// TIA Portal project "Project1" (V17)

(* hardware
DEVICE "S7-1200 station_1"  S7-1200 Station
   slot 0: "Rack_0"  S7-1200 Rack  Rack  V1.0
   slot 1: "PLC_1"  CPU 1214C DC/DC/DC  6ES7 214-1AG31-0XB0  V3.0
   slot 3: "AQ 1x12BIT_1"  AQ1 signal board  6ES7 232-4HA30-0XB0  V1.0
*)

// ===== PLC "PLC_1"  CPU 1214C DC/DC/DC =====

VAR_GLOBAL   // PLC tag table "Default tag table"
   "Carrega" AT %I0.0 : Bool;
   "Descarrega" AT %I0.1 : Bool;
   "MCarregando" AT %M0.0 : Bool;
   "MDescarregando" AT %M0.1 : Bool;
   "System_Byte" AT %MB6 : Byte;
   "FirstScan" AT %M6.0 : Bool;
   "DiagStatusUpdate" AT %M6.1 : Bool;
   "AlwaysTRUE" AT %M6.2 : Bool;
   "AlwaysFALSE" AT %M6.3 : Bool;
   "Clock_Byte" AT %MB5 : Byte;
   "Clock_10Hz" AT %M5.0 : Bool;
   "Clock_5Hz" AT %M5.1 : Bool;
   "Clock_2.5Hz" AT %M5.2 : Bool;
   "Clock_2Hz" AT %M5.3 : Bool;
   "Clock_1.25Hz" AT %M5.4 : Bool;
   "Clock_1Hz" AT %M5.5 : Bool;
   "Clock_0.625Hz" AT %M5.6 : Bool;
   "Clock_0.5Hz" AT %M5.7 : Bool;
   "System_Byte(1)" AT %MB5 : Byte;
   "LEDDescarga" AT %Q0.0 : Bool;
   "MCarregado" AT %M0.2 : Bool;
   "MDescarregado" AT %M0.3 : Bool;
   "LEDCarga" AT %Q0.1 : Bool;
   "Potenciometro" AT %IW64 : Int;
   "NORMEDPotenciometro" AT %MD100 : Real;
END_VAR

DATA_BLOCK "Data_block_1"   // DB2
{ S7_Optimized_Access := 'FALSE' }
VERSION : 0.1
   VAR
      ElipseCarregar : Bool;
      ElipseDescarregar : Bool;
      ElipsePotenciometro : Real;
   END_VAR
BEGIN
END_DATA_BLOCK

// folder: System blocks/Program resources

DATA_BLOCK "IEC_Counter_0_DB"   // DB1
{ S7_Optimized_Access := 'TRUE' }
AUTHOR : Simatic
FAMILY : IEC
NAME : CNTR
VERSION : 1.0
// stored: InstanceOfName IEC_COUNTER
"IEC_COUNTER"
BEGIN
END_DATA_BLOCK

// folder: (top level)

ORGANIZATION_BLOCK "Main"   // OB1, LAD, ProgramCycle
TITLE = "Main Program Sweep (Cycle)"
{ S7_Optimized_Access := 'TRUE' }
VERSION : 0.1
BEGIN

REGION Network 1
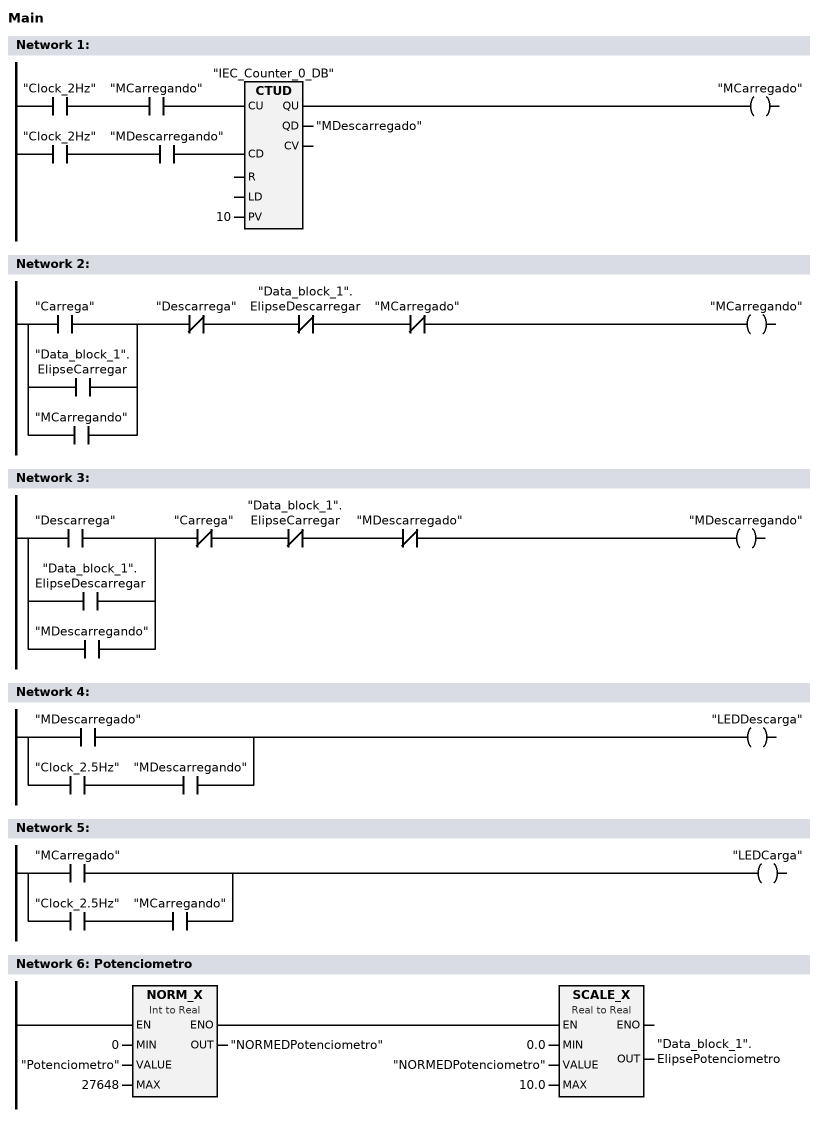
   "IEC_Counter_0_DB".CTUD(CU := "Clock_2Hz" AND "MCarregando",
                           CD := "Clock_2Hz" AND "MDescarregando",
                           PV := 10,
                           QD => "MDescarregado");
   "MCarregado" := "IEC_Counter_0_DB".QU;
END_REGION

REGION Network 2
   RUNG wire#powerrail
      Contact( "Carrega" )
      wire#w1
      I_Contact( "Descarrega" )
      I_Contact( "Data_block_1".ElipseDescarregar )
      I_Contact( "MCarregado" )
      Coil( "MCarregando" )
   END_RUNG
   RUNG wire#powerrail
      Contact( "Data_block_1".ElipseCarregar )
   END_RUNG wire#w1
   RUNG wire#powerrail
      Contact( "MCarregando" )
   END_RUNG wire#w1
   // the same network as SCL:
   "MCarregando" := ("Carrega" OR "Data_block_1".ElipseCarregar OR "MCarregando") AND NOT "Descarrega" AND NOT "Data_block_1".ElipseDescarregar AND NOT "MCarregado";
END_REGION

REGION Network 3
   RUNG wire#powerrail
      Contact( "Descarrega" )
      wire#w1
      I_Contact( "Carrega" )
      I_Contact( "Data_block_1".ElipseCarregar )
      I_Contact( "MDescarregado" )
      Coil( "MDescarregando" )
   END_RUNG
   RUNG wire#powerrail
      Contact( "Data_block_1".ElipseDescarregar )
   END_RUNG wire#w1
   RUNG wire#powerrail
      Contact( "MDescarregando" )
   END_RUNG wire#w1
   // the same network as SCL:
   "MDescarregando" := ("Descarrega" OR "Data_block_1".ElipseDescarregar OR "MDescarregando") AND NOT "Carrega" AND NOT "Data_block_1".ElipseCarregar AND NOT "MDescarregado";
END_REGION

REGION Network 4
   RUNG wire#powerrail
      Contact( "MDescarregado" )
      wire#w1
      Coil( "LEDDescarga" )
   END_RUNG
   RUNG wire#powerrail
      Contact( "Clock_2.5Hz" )
      Contact( "MDescarregando" )
   END_RUNG wire#w1
   // the same network as SCL:
   "LEDDescarga" := "MDescarregado" OR ("Clock_2.5Hz" AND "MDescarregando");
END_REGION

REGION Network 5
   RUNG wire#powerrail
      Contact( "MCarregado" )
      wire#w1
      Coil( "LEDCarga" )
   END_RUNG
   RUNG wire#powerrail
      Contact( "Clock_2.5Hz" )
      Contact( "MCarregando" )
   END_RUNG wire#w1
   // the same network as SCL:
   "LEDCarga" := "MCarregado" OR ("Clock_2.5Hz" AND "MCarregando");
END_REGION

REGION Network 6: Potenciometro
   RUNG wire#powerrail
      { S7_Templates := "[SrcType := Int, DestType := Real]"; S7_GenerateENO := "TRUE" } Normalize(min := 0, value := "Potenciometro", max := 27648, out => "NORMEDPotenciometro")
      { S7_Templates := "[SrcType := Real, DestType := Real]"; S7_GenerateENO := "TRUE" } Scale(min := 0.0, value := "NORMEDPotenciometro", max := 10.0, out => "Data_block_1".ElipsePotenciometro)
   END_RUNG
   // the same network as SCL:
   // ENO of a box is taken as its EN; it also drops when the box reports an error
   "NORMEDPotenciometro" := NORM_X(MIN := 0, VALUE := "Potenciometro", MAX := 27648);
   "Data_block_1".ElipsePotenciometro := SCALE_X(MIN := 0.0, VALUE := "NORMEDPotenciometro", MAX := 10.0);
END_REGION
END_ORGANIZATION_BLOCK